(* Logix 5000 project; controller chemical_plan vendor 1 type 14 code 150 rev 37.11; software revision 37.00 *)

TASK MainTask (continuous, watchdog 500 ms) : MainProgram

MODULES
   Local : vendor 1 type 14 code 150 (Compact 0, rev 37.11)
      Discrete_IO : Embedded (Compact 1, rev 3.1, Output RPI 20 ms)
      Analog_IO : Embedded (Compact 2, rev 1.1, Output RPI 80 ms)
      Counters : Embedded (Compact 3, rev 1.1, Output RPI 20 ms)
END_MODULES

VAR_GLOBAL   (* controller tags *)
   B11 : ALIAS FOR Local:1:I.Data.11;
   Drain_valve : ALIAS FOR Local:1:O.Data.10;
   Fillvalve : ALIAS FOR Local:2:O.Ch1Data;
   Height : REAL;
   HSC_CurrentCount : ALIAS FOR Local:3:I.Ctr0CurrentCount;
   HSC_Enable : ALIAS FOR Local:3:O.Ctr0En;
   HSC_Reset : ALIAS FOR Local:3:O.Ctr0SoftPreset;
   kFactor : DINT;
   Mixer : ALIAS FOR Local:1:O.Data.9;
   Pump : ALIAS FOR Local:1:O.Data.8;
   Seq1 : DINT;
   T1 : TIMER := (PRE := 1000);
   TargetTicks : DINT;
   TargetTicks90 : DINT;
   VallFull : DINT := 32000;
   VallQuarter : DINT := -20000;
   value : ALIAS FOR Local:2:I.Ch0Data;
   Valvehalf : DINT;
   zfh : DINT;
END_VAR

PROGRAM MainProgram   (* main routine MainRoutine *)

ROUTINE MainRoutine   (* ladder *)
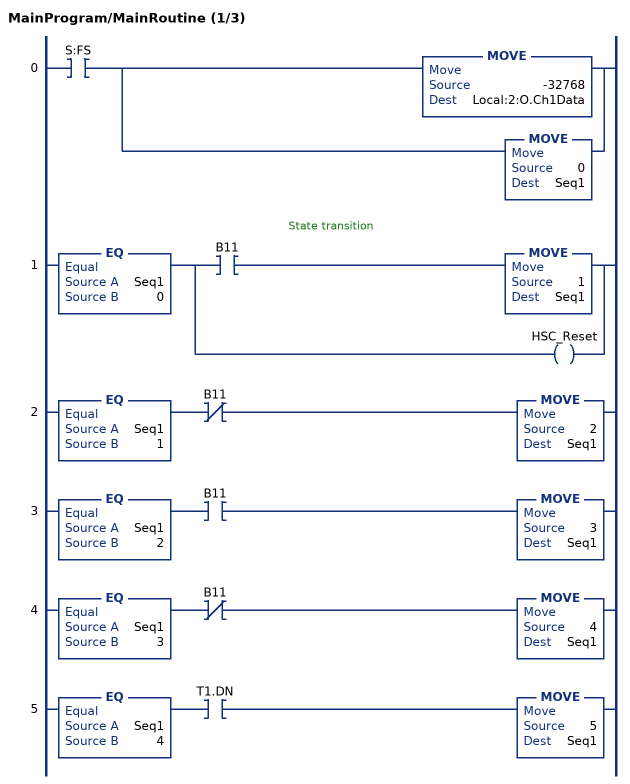
   0: XIC(S:FS)[MOVE(-32768,Local:2:O.Ch1Data) ,MOVE(0,Seq1) ];
   // State transition
   1: EQ(Seq1,0)[XIC(B11) MOVE(1,Seq1) ,OTE(HSC_Reset) ];
   2: EQ(Seq1,1)XIO(B11)MOVE(2,Seq1);
   3: EQ(Seq1,2)XIC(B11)MOVE(3,Seq1);
   4: EQ(Seq1,3)XIO(B11)MOVE(4,Seq1);
   5: EQ(Seq1,4)XIC(T1.DN)MOVE(5,Seq1);
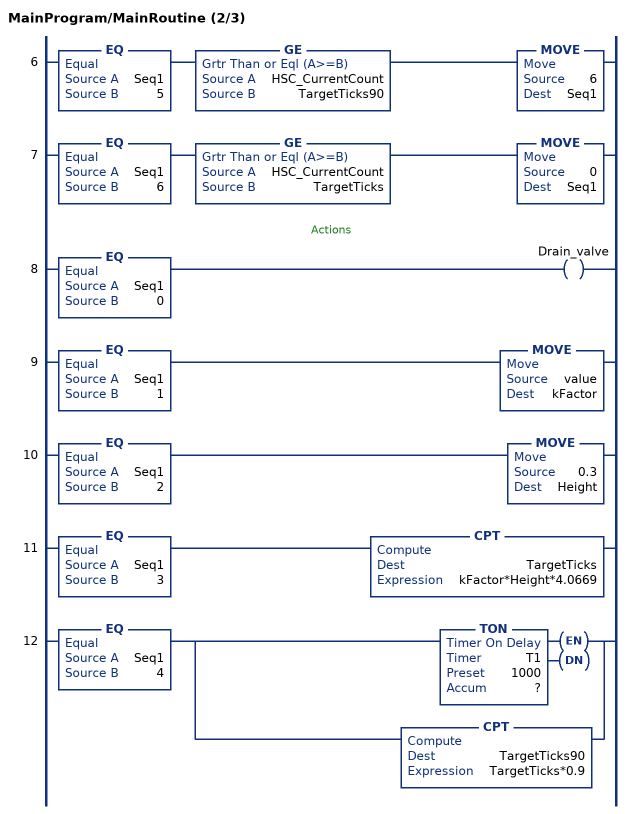
   6: EQ(Seq1,5)GE(HSC_CurrentCount,TargetTicks90)MOVE(6,Seq1);
   7: EQ(Seq1,6)GE(HSC_CurrentCount,TargetTicks)MOVE(0,Seq1);
   // Actions
   8: EQ(Seq1,0)OTE(Drain_valve);
   9: EQ(Seq1,1)MOVE(value,kFactor);
   10: EQ(Seq1,2)MOVE(0.3,Height);
   11: EQ(Seq1,3)CPT(TargetTicks,kFactor*Height*4.0669);
   12: EQ(Seq1,4)[TON(T1,?,?) ,CPT(TargetTicks90,TargetTicks*0.9) ];
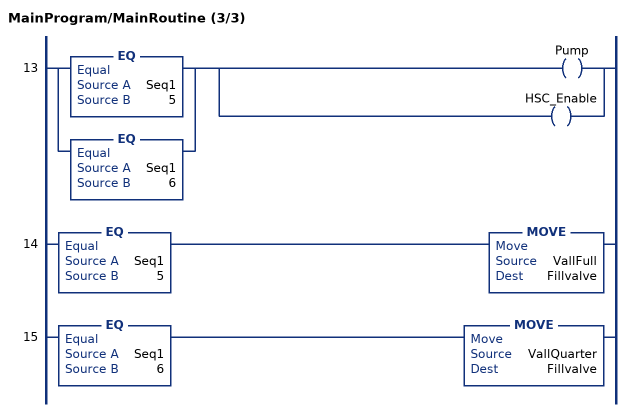
   13: [EQ(Seq1,5) ,EQ(Seq1,6) ][OTE(Pump) ,OTE(HSC_Enable) ];
   14: EQ(Seq1,5)MOVE(VallFull,Fillvalve);
   15: EQ(Seq1,6)MOVE(VallQuarter,Fillvalve);
END_ROUTINE
END_PROGRAM
